  (*-- TRANSITION --------------------------------------------------------------------------------------------------------------*)
  (*-- working folder not existing ------------------------------------------------------*)
  IF (_Active = FALSE)
  THEN
    _DeleteState:= E_TraceDeleteStates.WaitFolder;
  (*-- delay time over ------------------------------------------------------------------*)
  ELSIF(F_GetTimeMsDiff(_DeleteTime) >= T#10S)
  THEN
    _DeleteState:= E_TraceDeleteStates.FolderStart;
  END_IF




(********************************************************************************************************************************)
(** prepare folder scan *********************************************************************************************************)
E_TraceDeleteStates.FolderStart:
  (*-- ENTRY -------------------------------------------------------------------------------------------------------------------*)
  IF (_DeleteStateLast <> _DeleteState)
  THEN
    _DeleteStateLast:= _DeleteState;
    _DeleteTime     := F_GetTimeMsTick();
    (*-- prepare folder scan ------------------------------------------------------------*)
    _ScanSubFolder.eCmd:= E_EnumCmdType.eEnumCmd_First;
  END_IF

  (*-- ACTION ------------------------------------------------------------------------------------------------------------------*)

  (*-- TRANSITION --------------------------------------------------------------------------------------------------------------*)
    _DeleteState:= E_TraceDeleteStates.FolderSeek;




(********************************************************************************************************************************)
(** find next (sub) folder ******************************************************************************************************)
E_TraceDeleteStates.FolderSeek:
  (*-- ENTRY -------------------------------------------------------------------------------------------------------------------*)
  IF (_DeleteStateLast <> _DeleteState)
  THEN
    _DeleteStateLast:= _DeleteState;
    _DeleteTime     := F_GetTimeMsTick();
    (*-----------------------------------------------------------------------------------*)
    _ScanSubFolder( bExecute:= FALSE );
    _ScanSubFolder.sNetID   := '';   // local
//  _ScanSubFolder.eCmd;   (* hier nicht beschreiben *)
    _ScanSubFolder.bExecute := TRUE;
    _ScanSubFolder.tTimeout := Tc2_System.DEFAULT_ADS_TIMEOUT;
    (*-----------------------------------------------------------------------------------*)
    DestStart:= ADR(_ScanSubFolder.sPathName);
    DestEnd  := ADR(_ScanSubFolder.sPathName) + SIZEOF(_ScanSubFolder.sPathName);
    DestStart:= F_StringCopy( DestStart:= DestStart,  DestEnd:= DestEnd,  Source:= ADR(_MainFolder)  );
    DestStart:= F_StringCopy( DestStart:= DestStart,  DestEnd:= DestEnd,  Source:= ADR('/*.*')  );
  END_IF

  (*-- ACTION ------------------------------------------------------------------------------------------------------------------*)
  _ScanSubFolder();

  (*-- TRANSITION --------------------------------------------------------------------------------------------------------------*)
  IF (_ScanSubFolder.bBusy = FALSE)
  THEN
    _ScanSubFolder.eCmd:= E_EnumCmdType.eEnumCmd_Next;
    (*-- error --------------------------------------------------------------------------*)
    IF    (_ScanSubFolder.bError = TRUE)
    THEN  (* unfortunately no difference between path noch found or destination not reachable *)
      _DeleteState:= E_TraceDeleteStates.WaitDelay;
    (*-- folder completely scanned ------------------------------------------------------*)
    ELSIF (_ScanSubFolder.bEOE = TRUE)
    THEN
      _DeleteState:= E_TraceDeleteStates.WaitDelay;
    (*-- found entry is no folder => continue -------------------------------------------*)
    ELSIF (_ScanSubFolder.stFindFile.fileAttributes.bDirectory = FALSE)
    THEN
      _DeleteStateLast:= E_TraceDeleteStates.Initialization;   // Re-entry
    (*-- folder name invalid => continue ------------------------------------------------*)
    ELSIF (    (_ScanSubFolder.stFindFile.sFileName = '.' )
            OR (_ScanSubFolder.stFindFile.sFileName = '..')  )
    THEN
      _DeleteStateLast:= E_TraceDeleteStates.Initialization;   // Re-entry
    (*-- folder valid => old enough to delete? ------------------------------------------*)
    ELSE
      (*-- parse folder name according to 'YYYY-MM-DD' --------------*)
      Result:= F_StringToTimeDate( AllowInvalidChars:= FALSE,  // invalid charachters will lead to parsing error
                                   DestStart        := ADR(_ScanSubFolder.stFindFile.sFileName),
                                   DestEnd          := ADR(_ScanSubFolder.stFindFile.sFileName) + SIZEOF(_ScanSubFolder.stFindFile.sFileName),
                                   Result     => FolderDate  );
      (*-- calc difference (in ms due to TIME limitation of 42d) ----*)
      SystemTimeTD:= SYSTEMTIME_TO_DT(System.fbSystemTime.TIMESTR);
      FolderTimeTD:= SYSTEMTIME_TO_DT(FolderDate);
      Diff_Seconds:= DT_TO_LINT(SystemTimeTD) - DT_TO_LINT(FolderTimeTD);
     (*-- folder name doesnt fit naming scheme YYYY-MM-DD -----------*)
      IF (Result = FALSE)
      THEN  // ignore ==> continue
        _DeleteStateLast:= E_TraceDeleteStates.Initialization;   // Re-entry
      (*-- folder from future ;-) -----------------------------------*)
      ELSIF (Diff_Seconds < 0)
      THEN  // ignore ==> continue
        _DeleteStateLast:= E_TraceDeleteStates.Initialization;   // Re-entry
      (*-- folder according parsed name too old ---------------------*)
      ELSIF (Diff_Seconds * 1_000 >= TIME_TO_LINT(SHELF_LIFE)  )  // TIME is internally already ms
      THEN  // => empty and delete
        _DeleteState:= E_TraceDeleteStates.FileStart;
      (*-- keep searching -------------------------------------------*)
      ELSE
        _DeleteStateLast:= E_TraceDeleteStates.Initialization;   // Re-entry
      END_IF
    END_IF
  END_IF




(********************************************************************************************************************************)
(** prepare file scan ***********************************************************************************************************)
E_TraceDeleteStates.FileStart:
  (*-- ENTRY -------------------------------------------------------------------------------------------------------------------*)
  IF (_DeleteStateLast <> _DeleteState)
  THEN
    _DeleteStateLast:= _DeleteState;
    _DeleteTime     := F_GetTimeMsTick();
    (*-----------------------------------------------------------------------------------*)
    _FileFind.eCmd:= E_EnumCmdType.eEnumCmd_First;
  END_IF

  (*-- ACTION ------------------------------------------------------------------------------------------------------------------*)

  (*-- TRANSITION --------------------------------------------------------------------------------------------------------------*)
  _DeleteState:= E_TraceDeleteStates.FileSeek;




(********************************************************************************************************************************)
(** find a file *****************************************************************************************************************)
E_TraceDeleteStates.FileSeek:
  (*-- ENTRY -------------------------------------------------------------------------------------------------------------------*)
  IF (_DeleteStateLast <> _DeleteState)
  THEN
    _DeleteStateLast:= _DeleteState;
    _DeleteTime     := F_GetTimeMsTick();
    (*-----------------------------------------------------------------------------------*)
    _FileFind( bExecute:= FALSE );
    _FileFind.sNetID   := '';   // local
//  _FileFind.eCmd;      (* hier nicht beschreiben *)
    _FileFind.bExecute := TRUE;
    _FileFind.tTimeout := Tc2_System.DEFAULT_ADS_TIMEOUT;
    (*-----------------------------------------------------------------------------------*)
    DestStart:= ADR(_FileFind.sPathName);
    DestEnd  := ADR(_FileFind.sPathName) + SIZEOF(_FileFind.sPathName);
    DestStart:= F_StringCopy( DestStart:= DestStart,  DestEnd:= DestEnd,  Source:= ADR(_MainFolder)  );
    DestStart:= F_StringCopy( DestStart:= DestStart,  DestEnd:= DestEnd,  Source:= ADR('/')  );
    DestStart:= F_StringCopy( DestStart:= DestStart,  DestEnd:= DestEnd,  Source:= ADR(_ScanSubFolder.stFindFile.sFileName)  );
    DestStart:= F_StringCopy( DestStart:= DestStart,  DestEnd:= DestEnd,  Source:= ADR('/*.*')  );
  END_IF

  (*-- ACTION ------------------------------------------------------------------------------------------------------------------*)
  _FileFind();

  (*-- TRANSITION --------------------------------------------------------------------------------------------------------------*)
  IF ( _FileFind.bBusy = FALSE )
  THEN
    _FileFind.eCmd:= E_EnumCmdType.eEnumCmd_Next;
    (*-- error --------------------------------------------------------------------------*)
    IF    (_FileFind.bError = TRUE)
    THEN
      _DeleteState:= E_TraceDeleteStates.WaitDelay;
    (*-- folder completely scanned ------------------------------------------------------*)
    ELSIF (_FileFind.bEOE = TRUE)
    THEN
      _DeleteState:= E_TraceDeleteStates.FolderDelete;
    (*-- file name invalid => continue --------------------------------------------------*)
    ELSIF (    (_FileFind.stFindFile.sFileName = '.' )
            OR (_FileFind.stFindFile.sFileName = '..')  )
    THEN
      _DeleteStateLast:= E_TraceDeleteStates.Initialization;   // Re-entry
    (*-- file found ==> delete ----------------------------------------------------------*)
    ELSE
      _DeleteState:= E_TraceDeleteStates.FileDelete;
    END_IF
  END_IF




(********************************************************************************************************************************)
(** delete this one file ********************************************************************************************************)
E_TraceDeleteStates.FileDelete:
  (*-- ENTRY -------------------------------------------------------------------------------------------------------------------*)
  IF (_DeleteStateLast <> _DeleteState)
  THEN
    _DeleteStateLast:= _DeleteState;
    _DeleteTime     := F_GetTimeMsTick();
    (*-----------------------------------------------------------------------------------*)
    _FileDelete( bExecute:= FALSE );
    _FileDelete.sNetId   := '';   // local
    _FileDelete.ePath    := E_OpenPath.PATH_GENERIC;  
    _FileDelete.bExecute := TRUE;
    _FileDelete.tTimeout := Tc2_System.DEFAULT_ADS_TIMEOUT;               
    (*-----------------------------------------------------------------------------------*)
    DestStart:= ADR(_FileDelete.sPathName);
    DestEnd  := ADR(_FileDelete.sPathName) + SIZEOF(_FileDelete.sPathName);
    DestStart:= F_StringCopy( DestStart:= DestStart,  DestEnd:= DestEnd,  Source:= ADR(_MainFolder)  );
    DestStart:= F_StringCopy( DestStart:= DestStart,  DestEnd:= DestEnd,  Source:= ADR('/')  );
    DestStart:= F_StringCopy( DestStart:= DestStart,  DestEnd:= DestEnd,  Source:= ADR(_ScanSubFolder.stFindFile.sFileName)  );
    DestStart:= F_StringCopy( DestStart:= DestStart,  DestEnd:= DestEnd,  Source:= ADR('/')  );
    DestStart:= F_StringCopy( DestStart:= DestStart,  DestEnd:= DestEnd,  Source:= ADR(_FileFind.stFindFile.sFileName)  );
  END_IF

  (*-- ACTION ------------------------------------------------------------------------------------------------------------------*)
  _FileDelete();

  (*-- TRANSITION --------------------------------------------------------------------------------------------------------------*)
  IF ( _FileDelete.bBusy = FALSE )
  THEN
    _DeleteState:= E_TraceDeleteStates.FileSeek;
  END_IF




(********************************************************************************************************************************)
(** delete that (now empty) folder **********************************************************************************************)
E_TraceDeleteStates.FolderDelete:
  (*-- ENTRY -------------------------------------------------------------------------------------------------------------------*)
  IF (_DeleteStateLast <> _DeleteState)
  THEN
    _DeleteStateLast:= _DeleteState;
    _DeleteTime     := F_GetTimeMsTick();
    (*-----------------------------------------------------------------------------------*)
    _FolderRemove( bExecute:= FALSE );
    _FolderRemove.sNetId   := '';   // local
    _FolderRemove.ePath    := E_OpenPath.PATH_GENERIC;
    _FolderRemove.bExecute := TRUE;
    _FolderRemove.tTimeout := Tc2_System.DEFAULT_ADS_TIMEOUT;
    (*-----------------------------------------------------------------------------------*)
    DestStart:= ADR(_FolderRemove.sPathName);
    DestEnd  := ADR(_FolderRemove.sPathName) + SIZEOF(_FolderRemove.sPathName);
    DestStart:= F_StringCopy( DestStart:= DestStart,  DestEnd:= DestEnd,  Source:= ADR(_MainFolder)  );
    DestStart:= F_StringCopy( DestStart:= DestStart,  DestEnd:= DestEnd,  Source:= ADR('/')  );
    DestStart:= F_StringCopy( DestStart:= DestStart,  DestEnd:= DestEnd,  Source:= ADR(_ScanSubFolder.stFindFile.sFileName)  );
    DestStart:= F_StringCopy( DestStart:= DestStart,  DestEnd:= DestEnd,  Source:= ADR('/')  );
  END_IF

  (*-- ACTION ------------------------------------------------------------------------------------------------------------------*)
  _FolderRemove();

  (*-- TRANSITION --------------------------------------------------------------------------------------------------------------*)
  IF ( _FolderRemove.bBusy = FALSE )
  THEN
    _DeleteState:= E_TraceDeleteStates.HddUsage;
    (*-- trace it ---------------------------------------------------*)
// example: '11-000-0000-00-0, old folder deleted,  folder = D:/Traces/1979-01-09/'
    _Text:= '';
    _Text:= CONCAT(_Text, F_AddDividerToSisString(SubsystemRegistry.SubsystemName) );
    _Text:= CONCAT(_Text, ',  old folder deleted');
    _Text:= CONCAT(_Text, DebugTextBlocks.FOLDER);
    _Text:= CONCAT(_Text, _FolderRemove.sPathName);
    Put( MsgType := E_DebugMsgType.INFO,
         Instance:= ADR(_Instance),
         Text    := ADR(_Text)  );
  END_IF




(********************************************************************************************************************************)
(** read current hdd usage ******************************************************************************************************)
E_TraceDeleteStates.HddUsage:
  (*-- ENTRY -------------------------------------------------------------------------------------------------------------------*)
  IF (_DeleteStateLast <> _DeleteState)
  THEN
    _DeleteStateLast:= _DeleteState;
    _DeleteTime     := F_GetTimeMsTick();
    (*-----------------------------------------------------------------------------------*)
    _HddUsage.Start( Drive:= _MainFolder );  // use drive letter from main folder
  END_IF

  (*-- ACTION ------------------------------------------------------------------------------------------------------------------*)

  (*-- TRANSITION --------------------------------------------------------------------------------------------------------------*)
  IF (_HddUsage.Busy = FALSE)
  THEN
    _HddUsageCount:= _HddUsageCount + 1;
    _HddStateLast := E_TraceHddUsageStates.Initialization;  // force re-entry and write message
    (*-------------------------------------------*)
    _DeleteState:= E_TraceDeleteStates.FolderSeek;
  END_IF




(********************************************************************************************************************************)
(** unknown *********************************************************************************************************************)
ELSE
  _DeleteState:= E_TraceDeleteStates.Initialization;
END_CASE




(********************************************************************************************************************************)
(** done ************************************************************************************************************************)
END_METHOD

// creates hdd usage debug messages
METHOD PROTECTED M_RunHddUsage

(********************************************************************************************************************************)
VAR
END_VAR

(********************************************************************************************************************************)
(** diagnosis *******************************************************************************************************************)
{warning disable C0139}
_HddUsage.BytesTotal;
_HddUsage.BytesUsed;    _HddUsage.PercentageUsed;
_HddUsage.BytesFree;    _HddUsage.PercentageFree;
{warning restore C0139}




(********************************************************************************************************************************)
(** initialisation **************************************************************************************************************)
CASE (_HddState) OF
E_TraceHddUsageStates.Initialization:
  (*-- ENTRY -------------------------------------------------------------------------------------------------------------------*)
    _HddStateLast:= _HddState;
    _HddTooFull  := FALSE;

  (*-- ACTION ------------------------------------------------------------------------------------------------------------------*)

  (*-- TRANSITION --------------------------------------------------------------------------------------------------------------*)
    // takes place in state E_TraceCheckStates.HddUsage of M_RunCheck()




(********************************************************************************************************************************)
(** unknown *********************************************************************************************************************)
E_TraceHddUsageStates.Unknown:
  (*-- ENTRY -------------------------------------------------------------------------------------------------------------------*)
  IF (_HddStateLast <> _HddState)
  THEN
    _HddStateLast:= _HddState;
    _HddTooFull  := FALSE;
    (*-----------------------------------------------------------------------------------*)
    // example: '11-000-0000-00-0, unable to retrieve hdd usage,  drive = D:/'
    _Text:= '';
    _Text:= CONCAT(_Text, F_AddDividerToSisString(SubsystemRegistry.SubsystemName) );
    _Text:= CONCAT(_Text, ',  unable to retrieve hdd usage');
    _Text:= CONCAT(_Text, DebugTextBlocks.DRIVE);
    _Text:= CONCAT(_Text, _HddUsage.Drive);
    IF (_HddFullMissed <> 0)
    THEN
      _Text:= CONCAT(_Text, DebugTextBlocks.MISSED);  _Text:= CONCAT(_Text, ULINT_TO_STRING(_HddFullMissed)   );
    END_IF
    Put( MsgType := E_DebugMsgType.ERROR,
         Instance:= ADR(_Instance),
         Text    := ADR(_Text)  );
    (*-----------------------------------------------------------------------------------*)
    _HddFullMissed:= 0;
  END_IF

  (*-- ACTION ------------------------------------------------------------------------------------------------------------------*)

  (*-- TRANSITION --------------------------------------------------------------------------------------------------------------*)
    // takes place in state E_TraceCheckStates.HddUsage of M_RunCheck()




(********************************************************************************************************************************)
(** enough space free ***********************************************************************************************************)
E_TraceHddUsageStates.EnoughFree:
  (*-- ENTRY -------------------------------------------------------------------------------------------------------------------*)
  IF (_HddStateLast <> _HddState)
  THEN
    _HddStateLast:= _HddState;
    _HddTooFull  := FALSE;
    (*-----------------------------------------------------------------------------------*)
    // example: '11-000-0000-00-0, hdd usage information,  drive = D:/:,  total = 320GB,  free = 98GB,  usage = 65%'
    _Text:= '';
    _Text:= CONCAT(_Text, F_AddDividerToSisString(SubsystemRegistry.SubsystemName) );
    _Text:= CONCAT(_Text, ',  hdd usage information');
    _Text:= CONCAT(_Text, DebugTextBlocks.DRIVE);  _Text:= CONCAT(_Text, _HddUsage.Drive);
    _Text:= CONCAT(_Text, DebugTextBlocks.TOTAL);  _Text:= CONCAT(_Text, F_DiskSpaceToString(_HddUsage.BytesTotal)  );
    _Text:= CONCAT(_Text, DebugTextBlocks.FREE);   _Text:= CONCAT(_Text, F_DiskSpaceToString(_HddUsage.BytesFree)   );
    _Text:= CONCAT(_Text, DebugTextBlocks.USED);   _Text:= CONCAT(_Text, F_DiskSpaceToString(_HddUsage.BytesUsed)   );
    _Text:= CONCAT(_Text, DebugTextBlocks.USAGE);  _Text:= CONCAT(_Text, BYTE_TO_STRING(_HddUsage.PercentageUsed)   );  _Text:= CONCAT(_Text, '%');
    IF (_HddFullMissed <> 0)
    THEN
      _Text:= CONCAT(_Text, DebugTextBlocks.MISSED);  _Text:= CONCAT(_Text, ULINT_TO_STRING(_HddFullMissed)   );
    END_IF
    Put( MsgType := E_DebugMsgType.INFO,
         Instance:= ADR(_Instance),
         Text    := ADR(_Text)  );
    (*-----------------------------------------------------------------------------------*)
    _HddFullMissed:= 0;
  END_IF

  (*-- ACTION ------------------------------------------------------------------------------------------------------------------*)

  (*-- TRANSITION --------------------------------------------------------------------------------------------------------------*)
    // takes place in state E_TraceCheckStates.HddUsage of M_RunCheck()




(********************************************************************************************************************************)
(** warning level ***************************************************************************************************************)
E_TraceHddUsageStates.WarningLevel:
  (*-- ENTRY -------------------------------------------------------------------------------------------------------------------*)
  IF (_HddStateLast <> _HddState)
  THEN
    _HddStateLast:= _HddState;
    _HddTooFull  := FALSE;
    (*-----------------------------------------------------------------------------------*)
    // example: '11-000-0000-00-0, hdd usage information,  drive = D:/:,  total = 320GB,  free = 98GB,  usage = 65%,  missed messages = 1234'
    _Text:= '';
    _Text:= CONCAT(_Text, F_AddDividerToSisString(SubsystemRegistry.SubsystemName) );
    _Text:= CONCAT(_Text, ',  hdd usage information');
    _Text:= CONCAT(_Text, DebugTextBlocks.DRIVE);  _Text:= CONCAT(_Text, _HddUsage.Drive);
    _Text:= CONCAT(_Text, DebugTextBlocks.TOTAL);  _Text:= CONCAT(_Text, F_DiskSpaceToString(_HddUsage.BytesTotal)  );
    _Text:= CONCAT(_Text, DebugTextBlocks.FREE);   _Text:= CONCAT(_Text, F_DiskSpaceToString(_HddUsage.BytesFree)   );
    _Text:= CONCAT(_Text, DebugTextBlocks.USED);   _Text:= CONCAT(_Text, F_DiskSpaceToString(_HddUsage.BytesUsed)   );
    _Text:= CONCAT(_Text, DebugTextBlocks.USAGE);  _Text:= CONCAT(_Text, BYTE_TO_STRING(_HddUsage.PercentageUsed)   );  _Text:= CONCAT(_Text, '%');
    IF (_HddFullMissed <> 0)
    THEN
      _Text:= CONCAT(_Text, DebugTextBlocks.MISSED);  _Text:= CONCAT(_Text, ULINT_TO_STRING(_HddFullMissed)   );
    END_IF
    Put( MsgType := E_DebugMsgType.WARNING,
         Instance:= ADR(_Instance),
         Text    := ADR(_Text)  );
    (*-----------------------------------------------------------------------------------*)
    _HddFullMissed:= 0;
  END_IF

  (*-- ACTION ------------------------------------------------------------------------------------------------------------------*)

  (*-- TRANSITION --------------------------------------------------------------------------------------------------------------*)
    // takes place in state E_TraceCheckStates.HddUsage of M_RunCheck()




(********************************************************************************************************************************)
(** error level *****************************************************************************************************************)
E_TraceHddUsageStates.ErrorLevel:
  (*-- ENTRY -------------------------------------------------------------------------------------------------------------------*)
  IF (_HddStateLast <> _HddState)
  THEN
    _HddStateLast:= _HddState;
    (*-----------------------------------------------------------------------------------*)
    // example: '11-000-0000-00-0, hdd usage information,  drive = D:/:,  total = 320GB,  free = 98GB,  usage = 65%'
    _Text:= '';
    _Text:= CONCAT(_Text, F_AddDividerToSisString(SubsystemRegistry.SubsystemName) );
    _Text:= CONCAT(_Text, ',  hdd usage information');
    _Text:= CONCAT(_Text, DebugTextBlocks.DRIVE);  _Text:= CONCAT(_Text, _HddUsage.Drive);
    _Text:= CONCAT(_Text, DebugTextBlocks.TOTAL);  _Text:= CONCAT(_Text, F_DiskSpaceToString(_HddUsage.BytesTotal)  );
    _Text:= CONCAT(_Text, DebugTextBlocks.FREE);   _Text:= CONCAT(_Text, F_DiskSpaceToString(_HddUsage.BytesFree)   );
    _Text:= CONCAT(_Text, DebugTextBlocks.USED);   _Text:= CONCAT(_Text, F_DiskSpaceToString(_HddUsage.BytesUsed)   );
    _Text:= CONCAT(_Text, DebugTextBlocks.USAGE);  _Text:= CONCAT(_Text, BYTE_TO_STRING(_HddUsage.PercentageUsed)   );  _Text:= CONCAT(_Text, '%');
    Put( MsgType := E_DebugMsgType.ERROR,
         Instance:= ADR(_Instance),
         Text    := ADR(_Text)  );
    (*-----------------------------------------------------------------------------------*)
    _HddTooFull   := TRUE; // after this Put() just above
    _HddFullMissed:= 0;
  END_IF

  (*-- ACTION ------------------------------------------------------------------------------------------------------------------*)

  (*-- TRANSITION --------------------------------------------------------------------------------------------------------------*)
    // takes place in state E_TraceCheckStates.HddUsage of M_RunCheck()




(********************************************************************************************************************************)
(** unknown *********************************************************************************************************************)
ELSE
  _HddState:= E_TraceHddUsageStates.Initialization;
END_CASE




(********************************************************************************************************************************)
(** done ************************************************************************************************************************)
END_METHOD

// writes traces into file
METHOD PROTECTED M_RunWrite

(********************************************************************************************************************************)
VAR
  DestStart             : POINTER TO BYTE                  := 0;     // start position to concat
  DestEnd               : POINTER TO BYTE                  := 0;     // buffer/string end
END_VAR

(********************************************************************************************************************************)
(** initialization **************************************************************************************************************)
CASE(_WriteState) OF
E_TraceWriteStates.Initialization:
  (*-- ENTRY -------------------------------------------------------------------------------------------------------------------*)
    _WriteStateLast:= _WriteState;

  (*-- ACTION ------------------------------------------------------------------------------------------------------------------*)

  (*-- TRANSITION --------------------------------------------------------------------------------------------------------------*)
  _WriteState:= E_TraceWriteStates.WaitFolder;




(********************************************************************************************************************************)
(** error - wait to disable *****************************************************************************************************)
E_TraceWriteStates.Error:
  (*-- ENTRY -------------------------------------------------------------------------------------------------------------------*)
  IF (_WriteStateLast <> _WriteState)
  THEN
    _WriteStateLast:= _WriteState;
    _WriteTime     := F_GetTimeMsTick();
    (*-----------------------------------------------------------------------------------*)
  END_IF

  (*-- ACTION ------------------------------------------------------------------------------------------------------------------*)

  (*-- TRANSITION --------------------------------------------------------------------------------------------------------------*)
  (*-- working folder dissapeared -------------------------------------------------------*)
  IF (_Active = FALSE)
  THEN
    _WriteState:= E_TraceWriteStates.WaitFolder;
  END_IF




(********************************************************************************************************************************)
(** wait working folder *********************************************************************************************************)
E_TraceWriteStates.WaitFolder:
  (*-- ENTRY -------------------------------------------------------------------------------------------------------------------*)
  IF (_WriteStateLast <> _WriteState)
  THEN
    _WriteStateLast:= _WriteState;
    _WriteTime     := F_GetTimeMsTick();
    (*-----------------------------------------------------------------------------------*)
  END_IF

  (*-- ACTION ------------------------------------------------------------------------------------------------------------------*)

  (*-- TRANSITION --------------------------------------------------------------------------------------------------------------*)
  (*-- working folder exists ------------------------------------------------------------*)
  IF (_Active = TRUE)
  THEN
    _WriteState:= E_TraceWriteStates.StartWork;
  END_IF




(********************************************************************************************************************************)
(** build working folder name with date *****************************************************************************************)
E_TraceWriteStates.StartWork:
  (*-- ENTRY -------------------------------------------------------------------------------------------------------------------*)
  IF (_WriteStateLast <> _WriteState)
  THEN
    _WriteStateLast:= _WriteState;
    _WriteTime     := F_GetTimeMsTick();
    (*-- save current working date ------------------------------------------------------*)
    _WriteDate:= System.fbSystemTime.TIMESTR;
    (*-- build folder name --------------------------------------------------------------*)
    DestStart:= ADR(_WritePath);
    DestEnd  := ADR(_WritePath) + SIZEOF(_WritePath);
    DestStart:= F_StringCopy          ( DestStart:= DestStart,  DestEnd:= DestEnd,  Source    := ADR(_MainFolder)  );
    DestStart:= F_StringCopy          ( DestStart:= DestStart,  DestEnd:= DestEnd,  Source    := ADR('/')  );
    DestStart:= F_StringFromDatestruct( DestStart:= DestStart,  DestEnd:= DestEnd,  DateStruct:= _WriteDate );
    DestStart:= F_StringCopy          ( DestStart:= DestStart,  DestEnd:= DestEnd,  Source    := ADR('/')  );
  END_IF

  (*-- ACTION ------------------------------------------------------------------------------------------------------------------*)

  (*-- TRANSITION --------------------------------------------------------------------------------------------------------------*)
  _WriteState:= E_TraceWriteStates.CreateDir;




(********************************************************************************************************************************)
(** create daily working folder *************************************************************************************************)
E_TraceWriteStates.CreateDir:
  (*-- ENTRY -------------------------------------------------------------------------------------------------------------------*)
  IF (_WriteStateLast <> _WriteState)
  THEN
    _WriteStateLast:= _WriteState;
    _WriteTime     := F_GetTimeMsTick();
    (*-----------------------------------------------------------------------------------*)
    _CreateDir( bExecute:= FALSE );         
    _CreateDir.sNetId   := '';  // local
    _CreateDir.sPathName:= _WritePath;
    _CreateDir.ePath    := E_OpenPath.PATH_GENERIC;
    _CreateDir.bExecute := TRUE;         
    _CreateDir.tTimeout := Tc2_System.DEFAULT_ADS_TIMEOUT;
  END_IF

  (*-- ACTION ------------------------------------------------------------------------------------------------------------------*)
  _CreateDir();

  (*-- TRANSITION --------------------------------------------------------------------------------------------------------------*)
  IF (_CreateDir.bBusy = FALSE)
  THEN
    (*-- folder created => continue -----------------------------------------------------*)
    IF ( _CreateDir.bError = FALSE )
    THEN
      _WriteState:= E_TraceWriteStates.ScanFileStart;
      (*-- trace it -------------------------------------------------*)
// example: '11-000-0000-00-0, new folder created,  folder = D:/Traces/1979-01-09/'
      _Text:= '';
      _Text:= CONCAT(_Text, F_AddDividerToSisString(SubsystemRegistry.SubsystemName) );
      _Text:= CONCAT(_Text, ',  new folder created');
      _Text:= CONCAT(_Text, DebugTextBlocks.FOLDER);
      _Text:= CONCAT(_Text, _CreateDir.sPathName);
      Put( MsgType := E_DebugMsgType.INFO,
           Instance:= ADR(_Instance),
           Text    := ADR(_Text)  );
    (*-- folder already exists ----------------------------------------------------------*)
    ELSIF (    ( _CreateDir.nErrId = 16#070C )     // ADSERR_DEVICE_NOTFOUND
            OR ( _CreateDir.nErrId = 16#0723 )  )  // ADSERR_DEVICE_ACCESSDENIED
    THEN                                           // BKF-Flick: Änderung der ReturnCodes ab 4022.20
      _WriteState:= E_TraceWriteStates.ScanFileStart;
    (*-- error --------------------------------------------------------------------------*)
    ELSE
      _WriteState:= E_TraceWriteStates.Error;
    END_IF
  END_IF




(********************************************************************************************************************************)
(** prepare folder scan for existing files **************************************************************************************)
E_TraceWriteStates.ScanFileStart:
  (*-- ENTRY -------------------------------------------------------------------------------------------------------------------*)
  IF (_WriteStateLast <> _WriteState)
  THEN
    _WriteStateLast:= _WriteState;
    _WriteTime     := F_GetTimeMsTick();
    (*-----------------------------------------------------------------------------------*)
    _FileIndex     := 1;  (* Filenummerierung beginnt bei Eins *)
    _FileCheck.eCmd:= eEnumCmd_First;
  END_IF

  (*-- ACTION ------------------------------------------------------------------------------------------------------------------*)

  (*-- TRANSITION --------------------------------------------------------------------------------------------------------------*)
    _WriteState:= E_TraceWriteStates.ScanFileExists;




(********************************************************************************************************************************)
(** scan folder to check if files exist? ****************************************************************************************)
E_TraceWriteStates.ScanFileExists:
  (*-- ENTRY -------------------------------------------------------------------------------------------------------------------*)
  IF (_WriteStateLast <> _WriteState)
  THEN
    _WriteStateLast:= _WriteState;
    _WriteTime     := F_GetTimeMsTick();
    (*-- build file name with _FileIndex ------------------------------------------------*)
{warning disable C0139}
    M_BuildFileName();    _WriteFileName;
{warning restore C0139}
   (*-----------------------------------------------------------------------------------*)
    _FileCheck( bExecute:= FALSE );
    _FileCheck.sNetID   := '';  // local
//  _FileCheck.eCmd;   // maintain this value here 
    _FileCheck.bExecute := TRUE;
    _FileCheck.tTimeout := Tc2_System.DEFAULT_ADS_TIMEOUT;
    (*-----------------------------------------------------------------------------------*)
    DestStart:= ADR(_FileCheck.sPathName);
    DestEnd  := ADR(_FileCheck.sPathName) + SIZEOF(_FileCheck.sPathName);
    DestStart:= F_StringCopy( DestStart:= DestStart,  DestEnd:= DestEnd,  Source:= ADR(_WritePath)  );
    DestStart:= F_StringCopy( DestStart:= DestStart,  DestEnd:= DestEnd,  Source:= ADR(_WriteFileName)  );
  END_IF

  (*-- ACTION ------------------------------------------------------------------------------------------------------------------*)
  _FileCheck();

  (*-- TRANSITION --------------------------------------------------------------------------------------------------------------*)
  IF (_FileCheck.bBusy = FALSE)
  THEN
    _FileCheck.eCmd:= E_EnumCmdType.eEnumCmd_Next;
    (*-- error --------------------------------------------------------------------------*)
    IF ( _FileCheck.bError = TRUE )
    THEN
      _WriteState:= E_TraceWriteStates.Error;
    (*-- index does not exist => create & use -------------------------------------------*)
    ELSIF ( _FileCheck.bEOE = TRUE )
    THEN
      _WriteState:= E_TraceWriteStates.CreateOpen;
    (*-- found: but already too large => keep searching ---------------------------------*)
    ELSIF (    (_FileCheck.stFindFile.fileSize.dwLowPart)
            >= (_MaxFileSizeKB * DWORD#1024             )   ) (* kilo bytes => bytes *)
    THEN
      _WriteState:= E_TraceWriteStates.ScanFileCancel;
    (*-- found: smaller than max size => keep using -------------------------------------*)
    ELSE
      _WriteState:= E_TraceWriteStates.ScanFileAbort;
    END_IF
  END_IF




(********************************************************************************************************************************)
(** cancel scan *****************************************************************************************************************)
E_TraceWriteStates.ScanFileCancel:
  (*-- ENTRY -------------------------------------------------------------------------------------------------------------------*)
  IF (_WriteStateLast <> _WriteState)
  THEN
    _WriteStateLast:= _WriteState;
    _WriteTime     := F_GetTimeMsTick();
    (*-----------------------------------------------------------------------------------*)
    _FileCheck( bExecute:= FALSE );
    _FileCheck.sNetID   := '';  // local
//  _FileCheck.sPathName;  // maintain this value here 
    _FileCheck.eCmd     := E_EnumCmdType.eEnumCmd_Abort;
    _FileCheck.bExecute := TRUE;
    _FileCheck.tTimeout := Tc2_System.DEFAULT_ADS_TIMEOUT;
  END_IF

  (*-- ACTION ------------------------------------------------------------------------------------------------------------------*)
  _FileCheck();

  (*-- TRANSITION --------------------------------------------------------------------------------------------------------------*)
  IF (_FileCheck.bBusy = FALSE)
  THEN
    (*-- error --------------------------------------------------------------------------*)
    IF ( _FileCheck.bError = TRUE )
    THEN
      _WriteState:= E_TraceWriteStates.Error;
    (*-- cancellation successful --------------------------------------------------------*)
    ELSIF ( _FileCheck.bEOE = TRUE )
    THEN
      _FileIndex     := _FileIndex + 1;
      _FileCheck.eCmd:= eEnumCmd_First;
      _WriteState    := E_TraceWriteStates.ScanFileExists;
    (*-- keep searching -----------------------------------------------------------------*)
    ELSE
      _WriteStateLast:= E_TraceWriteStates.Initialization;  // Re-entry
    END_IF
  END_IF




(********************************************************************************************************************************)
(** cancel scan *****************************************************************************************************************)
E_TraceWriteStates.ScanFileAbort:
  (*-- ENTRY -------------------------------------------------------------------------------------------------------------------*)
  IF (_WriteStateLast <> _WriteState)
  THEN
    _WriteStateLast:= _WriteState;
    _WriteTime     := F_GetTimeMsTick();
    (*-----------------------------------------------------------------------------------*)
    _FileCheck( bExecute:= FALSE );
    _FileCheck.sNetID   := '';  // local
//  _FileCheck.sPathName;  // maintain this value here 
    _FileCheck.eCmd     := E_EnumCmdType.eEnumCmd_Abort;
    _FileCheck.bExecute := TRUE;
    _FileCheck.tTimeout := Tc2_System.DEFAULT_ADS_TIMEOUT;
  END_IF

  (*-- ACTION ------------------------------------------------------------------------------------------------------------------*)
  _FileCheck();

  (*-- TRANSITION --------------------------------------------------------------------------------------------------------------*)
  IF (_FileCheck.bBusy = FALSE)
  THEN
    (*-- error --------------------------------------------------------------------------*)
    IF    ( _FileCheck.bError = TRUE )
    THEN
      _WriteState:= E_TraceWriteStates.Error;
    (*-- cancellation successful --------------------------------------------------------*)
    ELSIF ( _FileCheck.bEOE = TRUE )
    THEN
      _WriteState:= E_TraceWriteStates.WaitForTrace;
    (*-- keep searching -----------------------------------------------------------------*)
    ELSE                                     
      _WriteStateLast:= E_TraceWriteStates.Initialization;  // Re-entry
    END_IF
  END_IF




(********************************************************************************************************************************)
(** create new file *************************************************************************************************************)
E_TraceWriteStates.CreateOpen:
  (*-- ENTRY -------------------------------------------------------------------------------------------------------------------*)
  IF (_WriteStateLast <> _WriteState)
  THEN
    _WriteStateLast:= _WriteState;
    _WriteTime     := F_GetTimeMsTick();
    (*-- build file name with _FileIndex ------------------------------------------------*)
{warning disable C0139}
    M_BuildFileName();    _WriteFileName;
{warning restore C0139}
    (*-----------------------------------------------------------------------------------*)
    _FileOpen( bExecute:= FALSE );
    _FileOpen.sNetId   := '';  // local
    _FileOpen.nMode    := ( FOPEN_MODEWRITE OR FOPEN_MODEPLUS OR FOPEN_MODEBINARY );
    _FileOpen.ePath    := E_OpenPath.PATH_GENERIC;          
    _FileOpen.bExecute := TRUE;
    _FileOpen.tTimeout := Tc2_System.DEFAULT_ADS_TIMEOUT;
    (*-----------------------------------------------------------------------------------*)
    DestStart:= ADR(_FileOpen.sPathName);
    DestEnd  := ADR(_FileOpen.sPathName) + SIZEOF(_FileOpen.sPathName);
    DestStart:= F_StringCopy( DestStart:= DestStart,  DestEnd:= DestEnd,  Source:= ADR(_WritePath)  );
    DestStart:= F_StringCopy( DestStart:= DestStart,  DestEnd:= DestEnd,  Source:= ADR(_WriteFileName)  );
  END_IF

  (*-- ACTION ------------------------------------------------------------------------------------------------------------------*)
  _FileOpen();

  (*-- TRANSITION --------------------------------------------------------------------------------------------------------------*)
  IF (_FileOpen.bBusy = FALSE)
  THEN
    (*-- File angelegt ------------------------------------------------------------------*)
    IF    ( _FileOpen.bError = FALSE )  
    THEN
      _Statistics.FileOpenCounter:= _Statistics.FileOpenCounter + 1;
      (*-----------------------------------------*)
      _Opened        := TRUE;
      _FileTimeOpened:= F_GetTimeMsTick();
      _WriteState    := E_TraceWriteStates.CreateHeader;
   (*-- folder doesn't exist (anymore) --------------------------------------------------*)
    ELSIF ( _FileOpen.nErrId = 16#070C )
    THEN
      _WriteState:= E_TraceWriteStates.StartWork;    
    (*-- error --------------------------------------------------------------------------*)
    ELSE
      _WriteState:= E_TraceWriteStates.Error;
    END_IF
  END_IF




(********************************************************************************************************************************)
(** write header ****************************************************************************************************************)
E_TraceWriteStates.CreateHeader:
  (*-- ENTRY -------------------------------------------------------------------------------------------------------------------*)
  IF (_WriteStateLast <> _WriteState)
  THEN
    _WriteStateLast:= _WriteState;
    _WriteTime     := F_GetTimeMsTick();
    (*-- create file header -------------------------------------------------------------*)
{warning disable C0139}
    M_CreateHeader();   _DataLength;
{warning restore C0139}
    (*-----------------------------------------------------------------------------------*)
    _FileWrite( bExecute:= FALSE );
    _FileWrite.sNetId    := '';  // local               
    _FileWrite.hFile     := _FileOpen.hFile;       
    _FileWrite.pWriteBuff:= ADR(_DataBuffer);
    _FileWrite.cbWriteLen:= _DataLength;
    _FileWrite.bExecute  := TRUE;
    _FileWrite.tTimeout  := Tc2_System.DEFAULT_ADS_TIMEOUT;
  END_IF

  (*-- ACTION ------------------------------------------------------------------------------------------------------------------*)
  _FileWrite();

  (*-- TRANSITION --------------------------------------------------------------------------------------------------------------*)
  IF (_FileWrite.bBusy = FALSE)
  THEN
    (*-- error --------------------------------------------------------------------------*)
    IF    ( _FileWrite.bError = TRUE )
    THEN
      _WriteState:= E_TraceWriteStates.Error;
    (*-- writing successful -------------------------------------------------------------*)
    ELSE
      _WriteState:= E_TraceWriteStates.CreateClose;
    END_IF
  END_IF




(********************************************************************************************************************************)
(** close new file **************************************************************************************************************)
E_TraceWriteStates.CreateClose:
  (*-- ENTRY -------------------------------------------------------------------------------------------------------------------*)
  IF (_WriteStateLast <> _WriteState)
  THEN
    _WriteStateLast:= _WriteState;
    _WriteTime     := F_GetTimeMsTick();
    (*-----------------------------------------------------------------------------------*)
    _FileClose( bExecute:= FALSE );
    _FileClose.sNetId  := '';   // local
    _FileClose.hFile   := _FileOpen.hFile;
    _FileClose.bExecute:= TRUE;
    _FileClose.tTimeout:= Tc2_System.DEFAULT_ADS_TIMEOUT;
  END_IF

  (*-- ACTION ------------------------------------------------------------------------------------------------------------------*)
  _FileClose();

  (*-- TRANSITION --------------------------------------------------------------------------------------------------------------*)
  IF (_FileClose.bBusy = FALSE)
  THEN
    _PlcRestarted:= FALSE;
    _Opened      := FALSE;
    (*-- calculate maximum file open time -----------------------------------------------*)
    _Statistics.MaxFileOpenTime:= MAX( _Statistics.MaxFileOpenTime, F_GetTimeMsDiff(_FileTimeOpened)  );
    (*-- error --------------------------------------------------------------------------*)
    IF    ( _FileClose.bError = TRUE )
    THEN
      _WriteState:= E_TraceWriteStates.Error;
    (*-- closing successful -------------------------------------------------------------*)
    ELSE
      _WriteState:= E_TraceWriteStates.WaitForTrace;
    END_IF
  END_IF




(********************************************************************************************************************************)
(** inhibit time (currently not used) *******************************************************************************************)
E_TraceWriteStates.WaitLocked:
  (*-- ENTRY -------------------------------------------------------------------------------------------------------------------*)
  IF (_WriteStateLast <> _WriteState)
  THEN
    _WriteStateLast:= _WriteState;
    _WriteTime     := F_GetTimeMsTick();
    (*-----------------------------------------------------------------------------------*)
  END_IF

  (*-- ACTION ------------------------------------------------------------------------------------------------------------------*)

  (*-- TRANSITION --------------------------------------------------------------------------------------------------------------*)
  (*-- (still) too many traces to be written -> skip inhibit time -----------------------*)
  IF (_FifoFillLevel >= 256)
  THEN
    _WriteState:= E_TraceWriteStates.WaitForTrace;
  (*-- inhibit time over ----------------------------------------------------------------*)
  ELSIF (F_GetTimeMsDiff(_WriteTime) >= LOCKTIME)
  THEN
    _WriteState:= E_TraceWriteStates.WaitForTrace;
  (*-- working folder dissapeared -------------------------------------------------------*)
  ELSIF (_Active = FALSE)
  THEN
    _WriteState:= E_TraceWriteStates.WaitFolder;
  END_IF




(********************************************************************************************************************************)
(** idle -> wait for traces to write ********************************************************************************************)
E_TraceWriteStates.WaitForTrace:
  (*-- ENTRY -------------------------------------------------------------------------------------------------------------------*)
  IF (_WriteStateLast <> _WriteState)
  THEN
    _WriteStateLast:= _WriteState;
    _WriteTime     := F_GetTimeMsTick();
    (*-----------------------------------------------------------------------------------*)
  END_IF

  (*-- ACTION ------------------------------------------------------------------------------------------------------------------*)

  (*-- TRANSITION --------------------------------------------------------------------------------------------------------------*)
  (*-- traces to write available --------------------------------------------------------*)
  IF (_FifoFillLevel <> 0)
  THEN
//  IF ( _FileIndex <> 1 ) 
//  THEN
//     => check if file-one (still) exists
//  ELSE
    _FileCheck.eCmd:= E_EnumCmdType.eEnumCmd_First;
    _WriteState    := E_TraceWriteStates.FileSizeExists;
  (*-- working folder dissapeared -------------------------------------------------------*)
  ELSIF (_Active = FALSE)
  THEN
    _WriteState:= E_TraceWriteStates.WaitFolder;
  END_IF




(********************************************************************************************************************************)
(** check if current file (_FileIndex) still exists and if it's (already) too large *********************************************)
E_TraceWriteStates.FileSizeExists:
  (*-- ENTRY -------------------------------------------------------------------------------------------------------------------*)
  IF (_WriteStateLast <> _WriteState)
  THEN
    _WriteStateLast:= _WriteState;
    _WriteTime     := F_GetTimeMsTick();
    (*-----------------------------------------------------------------------------------*)
    _FileCheck( bExecute:= FALSE );
    _FileCheck.sNetID   := '';   // local
//  _FileCheck.eCmd;   (* nicht beschreiben *)
    _FileCheck.bExecute := TRUE;
    _FileCheck.tTimeout := Tc2_System.DEFAULT_ADS_TIMEOUT;
    (*-----------------------------------------------------------------------------------*)
    DestStart:= ADR(_FileCheck.sPathName);
    DestEnd  := ADR(_FileCheck.sPathName) + SIZEOF(_FileCheck.sPathName);
    DestStart:= F_StringCopy( DestStart:= DestStart,  DestEnd:= DestEnd,  Source:= ADR(_WritePath)  );
    DestStart:= F_StringCopy( DestStart:= DestStart,  DestEnd:= DestEnd,  Source:= ADR(_WriteFileName)  );
  END_IF

  (*-- ACTION ------------------------------------------------------------------------------------------------------------------*)
  _FileCheck();

  (*-- TRANSITION --------------------------------------------------------------------------------------------------------------*)
  IF (_FileCheck.bBusy = FALSE)
  THEN
    (*-- error --------------------------------------------------------------------------*)
    IF    (_FileCheck.bError = TRUE)
    THEN
      _WriteState:= E_TraceWriteStates.Error;
    (*-- doesnt exists (anymore) => rescan ----------------------------------------------*)
    ELSIF (_FileCheck.bEOE = TRUE)
    THEN
      _WriteState:= E_TraceWriteStates.ScanFileStart;
    (*-- exists: => use it --------------------------------------------------------------*)
    ELSE
      _FileSize  := (        DWORD_TO_ULINT(_FileCheck.stFindFile.fileSize.dwLowPart )
                      OR SHL(DWORD_TO_ULINT(_FileCheck.stFindFile.fileSize.dwHighPart), 32)  );
      (*-- maximal file size exceeded -----------*)
      IF (    (_FileSize (* KiloBytes => Bytes *) )
           >= (_MaxFileSizeKB * ULINT#1024        )   )  THEN   _WriteState:= E_TraceWriteStates.FileSizeCancel;  // start over with new file index
      ELSE                                                      _WriteState:= E_TraceWriteStates.FileSizeAbort;   // use this file again
      END_IF
    END_IF
  END_IF




(********************************************************************************************************************************)
(** cancel file size/exist check and use this ***********************************************************************************)
E_TraceWriteStates.FileSizeAbort:
  (*-- ENTRY -------------------------------------------------------------------------------------------------------------------*)
  IF (_WriteStateLast <> _WriteState)
  THEN
    _WriteStateLast:= _WriteState;
    _WriteTime     := F_GetTimeMsTick();
    (*-----------------------------------------------------------------------------------*)
    _FileCheck( bExecute:= FALSE );
    _FileCheck.sNetID   := '';   // local
//  _FileCheck.sPathName;  remain value
    _FileCheck.eCmd     := E_EnumCmdType.eEnumCmd_Abort;
    _FileCheck.bExecute := TRUE;
    _FileCheck.tTimeout := Tc2_System.DEFAULT_ADS_TIMEOUT;
  END_IF

  (*-- ACTION ------------------------------------------------------------------------------------------------------------------*)
  _FileCheck();

  (*-- TRANSITION --------------------------------------------------------------------------------------------------------------*)
  IF ( _FileCheck.bBusy = FALSE )
  THEN
    (*-- error --------------------------------------------------------------------------*)
    IF    (_FileCheck.bError = TRUE)
    THEN
      _WriteState:= E_TraceWriteStates.Error;
    (*-- finished -----------------------------------------------------------------------*)
    ELSIF (_FileCheck.bEOE = TRUE)
    THEN
      _WriteState:= E_TraceWriteStates.OpenAppend;
    (*-- keep searching -----------------------------------------------------------------*)
    ELSE
      _WriteStateLast:= E_TraceWriteStates.Initialization;  // Re-entry
    END_IF
  END_IF



(********************************************************************************************************************************)
(** cancel file size/exist check due to file size already too large *************************************************************)
E_TraceWriteStates.FileSizeCancel:
  (*-- ENTRY -------------------------------------------------------------------------------------------------------------------*)
  IF (_WriteStateLast <> _WriteState)
  THEN
    _WriteStateLast:= _WriteState;
    _WriteTime     := F_GetTimeMsTick();
    (*-----------------------------------------------------------------------------------*)
    _FileCheck( bExecute:= FALSE );
    _FileCheck.sNetID   := '';   // local
//  _FileCheck.sPathName;  remain value
    _FileCheck.eCmd     := E_EnumCmdType.eEnumCmd_Abort;
    _FileCheck.bExecute := TRUE;
    _FileCheck.tTimeout := Tc2_System.DEFAULT_ADS_TIMEOUT;
  END_IF

  (*-- ACTION ------------------------------------------------------------------------------------------------------------------*)
  _FileCheck();

  (*-- TRANSITION --------------------------------------------------------------------------------------------------------------*)
  IF ( _FileCheck.bBusy = FALSE )
  THEN
    (*-- error --------------------------------------------------------------------------*)
    IF    (_FileCheck.bError = TRUE)
    THEN
      _WriteState:= E_TraceWriteStates.Error;
    (*-- finished -----------------------------------------------------------------------*)
    ELSIF (_FileCheck.bEOE = TRUE)
    THEN
      _FileIndex := _FileIndex + 1;
      _WriteState:= E_TraceWriteStates.CreateOpen;
    (*-- keep searching -----------------------------------------------------------------*)
    ELSE
      _WriteStateLast:= E_TraceWriteStates.Initialization;  // Re-entry
    END_IF
  END_IF




(********************************************************************************************************************************)
(** open file to write/append ***************************************************************************************************)
E_TraceWriteStates.OpenAppend:
  (*-- ENTRY -------------------------------------------------------------------------------------------------------------------*)
  IF (_WriteStateLast <> _WriteState)
  THEN
    _WriteStateLast:= _WriteState;
    _WriteTime     := F_GetTimeMsTick();
    (*-----------------------------------------------------------------------------------*)
    _FileOpen( bExecute:= FALSE );
    _FileOpen.sNetId   := '';   // local
    _FileOpen.nMode    := ( FOPEN_MODEAPPEND OR FOPEN_MODEBINARY );                                
    _FileOpen.ePath    := E_OpenPath.PATH_GENERIC;          
    _FileOpen.bExecute := TRUE;
    _FileOpen.tTimeout := Tc2_System.DEFAULT_ADS_TIMEOUT;
    (*-----------------------------------------------------------------------------------*)
    DestStart:= ADR(_FileOpen.sPathName);
    DestEnd  := ADR(_FileOpen.sPathName) + SIZEOF(_FileOpen.sPathName);
    DestStart:= F_StringCopy( DestStart:= DestStart,  DestEnd:= DestEnd,  Source:= ADR(_WritePath)  );
    DestStart:= F_StringCopy( DestStart:= DestStart,  DestEnd:= DestEnd,  Source:= ADR(_WriteFileName)  );
  END_IF

  (*-- ACTION ------------------------------------------------------------------------------------------------------------------*)
  _FileOpen();

  (*-- TRANSITION --------------------------------------------------------------------------------------------------------------*)
  IF ( _FileOpen.bBusy = FALSE )
  THEN
    (*-- file opened --------------------------------------------------------------------*)
    IF    ( _FileOpen.bError = FALSE )  
    THEN
      _Statistics.FileOpenCounter:= _Statistics.FileOpenCounter + 1;
      _FileTimeOpened            := F_GetTimeMsTick();
      _Opened                    := TRUE;
      (*-----------------------------------------*)
      IF (_PlcRestarted = TRUE) THEN   _WriteState:= E_TraceWriteStates.WriteDivider;
      ELSE                             _WriteState:= E_TraceWriteStates.WriteData;
      END_IF
    (*-- folder doesn't exist (anymore) -------------------------------------------------*)
    ELSIF ( _FileOpen.nErrId = 16#070C )
    THEN
      _WriteState:= E_TraceWriteStates.StartWork;    
    (*-- error --------------------------------------------------------------------------*)
    ELSE
      _WriteState:= E_TraceWriteStates.Error;
    END_IF
  END_IF




(********************************************************************************************************************************)
(** add plc restart divider *****************************************************************************************************)
E_TraceWriteStates.WriteDivider:
  (*-- ENTRY -------------------------------------------------------------------------------------------------------------------*)
  IF (_WriteStateLast <> _WriteState)
  THEN
    _WriteStateLast:= _WriteState;
    _WriteTime     := F_GetTimeMsTick();
    (*-- create plc divider -------------------------------------------------------------*)
{warning disable C0139}
    M_CreatePlcDivider();   _DataLength;
{warning restore C0139}
    (*-----------------------------------------------------------------------------------*)
    _FileWrite( bExecute:= FALSE );
    _FileWrite.sNetId    := '';  // local               
    _FileWrite.hFile     := _FileOpen.hFile;       
    _FileWrite.pWriteBuff:= ADR(_DataBuffer);
    _FileWrite.cbWriteLen:= _DataLength;
    _FileWrite.bExecute  := TRUE;
    _FileWrite.tTimeout  := Tc2_System.DEFAULT_ADS_TIMEOUT;
  END_IF

  (*-- ACTION ------------------------------------------------------------------------------------------------------------------*)
  _FileWrite();

  (*-- TRANSITION --------------------------------------------------------------------------------------------------------------*)
  IF (_FileWrite.bBusy = FALSE)
  THEN
    _PlcRestarted:= FALSE;
    _FileSize    := _FileSize + _FileWrite.cbWrite;
    (*-- error --------------------------------------------------------------------------*)
    IF    (_FileWrite.bError = TRUE)
    THEN
      _WriteState:= E_TraceWriteStates.CloseOpenTime;
    (*-- writing successful -------------------------------------------------------------*)
    ELSE
      _WriteState:= E_TraceWriteStates.WriteData;
    END_IF
  END_IF




(********************************************************************************************************************************)
(** write trace lines ***********************************************************************************************************)
E_TraceWriteStates.WriteData:
  (*-- ENTRY -------------------------------------------------------------------------------------------------------------------*)
  IF (_WriteStateLast <> _WriteState)
  THEN
    _WriteStateLast:= _WriteState;
    _WriteTime     := F_GetTimeMsTick();
    (*-- create data --------------------------------------------------------------------*)
{warning disable C0139}
    _DataDateChanged:= M_CreateData();   _DataLength;
    (*-----------------------------------------------------------------------------------*)
    _FileWrite( bExecute:= FALSE );
    _FileWrite.sNetId    := '';  // local               
    _FileWrite.hFile     := _FileOpen.hFile;       
    _FileWrite.pWriteBuff:= ADR(_DataBuffer);
    _FileWrite.cbWriteLen:= _DataLength;
    _FileWrite.bExecute  := TRUE;
    _FileWrite.tTimeout  := Tc2_System.DEFAULT_ADS_TIMEOUT;
{warning restore C0139}
  END_IF

  (*-- ACTION ------------------------------------------------------------------------------------------------------------------*)
  _FileWrite();

  (*-- TRANSITION --------------------------------------------------------------------------------------------------------------*)
  IF ( _FileWrite.bBusy = FALSE )
  THEN
    _FileSize:= _FileSize + _FileWrite.cbWrite;
    (*-- error --------------------------------------------------------------------------*)
    IF    (_FileWrite.bError = TRUE)
    THEN
      _WriteState:= E_TraceWriteStates.CloseOpenTime;
    (*-- trace date changed -> new date folder ------------------------------------------*)
    ELSIF (_DataDateChanged = TRUE)
    THEN  (* new file/folder for new day *)
      _WriteState:= E_TraceWriteStates.EofDate;
    (*-- maximum file size exceeded -----------------------------------------------------*)
    ELSIF (    (_FileSize (* KiloBytes => Bytes *) )
            >= (_MaxFileSizeKB * ULINT#1024        )   )
    THEN  (* start over with new file index *)
      _WriteState:= E_TraceWriteStates.EofSize;
    (*-- maximum file open time exceeded (flush) ----------------------------------------*)
    ELSIF (F_GetTimeMsDiff(_FileTimeOpened) >= MAX_FILEOPEN_TIME)
    THEN  (* close file and re-open it => file flush *)
      _WriteState:= E_TraceWriteStates.CloseOpenTime;
    (*-- more to write? -----------------------------------------------------------------*)
    ELSIF (_FifoFillLevel <> 0)
    THEN
      _WriteStateLast:= E_TraceWriteStates.Initialization;  // Re-entry
    (*-- no traces to write anymore -> close & wait -------------------------------------*)
    ELSE
      _WriteState:= E_TraceWriteStates.CloseOpenTime;
    END_IF
  END_IF




(********************************************************************************************************************************)
(** close due to max open time exceeded *****************************************************************************************)
E_TraceWriteStates.CloseOpenTime:
  (*-- ENTRY -------------------------------------------------------------------------------------------------------------------*)
  IF (_WriteStateLast <> _WriteState)
  THEN
    _WriteStateLast:= _WriteState;
    _WriteTime     := F_GetTimeMsTick();
    (*-----------------------------------------------------------------------------------*)
    _FileClose( bExecute:= FALSE );
    _FileClose.sNetId  := '';  // local
    _FileClose.hFile   := _FileOpen.hFile;
    _FileClose.bExecute:= TRUE;
    _FileClose.tTimeout:= Tc2_System.DEFAULT_ADS_TIMEOUT;
  END_IF

  (*-- ACTION ------------------------------------------------------------------------------------------------------------------*)
  _FileClose();

  (*-- TRANSITION --------------------------------------------------------------------------------------------------------------*)
  IF (_FileClose.bBusy = FALSE)
  THEN
    _Opened:= FALSE;
    (*-- calculate maximum file open time -----------------------------------------------*)
    _Statistics.MaxFileOpenTime:= MAX( _Statistics.MaxFileOpenTime, F_GetTimeMsDiff(_FileTimeOpened)  );
    (*-- error --------------------------------------------------------------------------*)
    IF    (_FileClose.bError = TRUE)
    THEN
      _WriteState:= E_TraceWriteStates.Error;
    (*-- closing successful -------------------------------------------------------------*)
    ELSE
      _WriteState:= E_TraceWriteStates.WaitLocked;
    END_IF
  END_IF




(********************************************************************************************************************************)
(** add eof due max file size exceeded ******************************************************************************************)
E_TraceWriteStates.EofSize:
  (*-- ENTRY -------------------------------------------------------------------------------------------------------------------*)
  IF (_WriteStateLast <> _WriteState)
  THEN
    _WriteStateLast:= _WriteState;
    _WriteTime     := F_GetTimeMsTick();
    (*-- create eof ---------------------------------------------------------------------*)
{warning disable C0139}
    M_CreateEof();   _DataLength;
{warning restore C0139}
    (*-----------------------------------------------------------------------------------*)
    _FileWrite( bExecute:= FALSE );
    _FileWrite.sNetId    := '';  // local               
    _FileWrite.hFile     := _FileOpen.hFile;       
    _FileWrite.pWriteBuff:= ADR(_DataBuffer);
    _FileWrite.cbWriteLen:= _DataLength;
    _FileWrite.bExecute  := TRUE;
    _FileWrite.tTimeout  := Tc2_System.DEFAULT_ADS_TIMEOUT;
  END_IF

  (*-- ACTION ------------------------------------------------------------------------------------------------------------------*)
  _FileWrite();

  (*-- TRANSITION --------------------------------------------------------------------------------------------------------------*)
  IF (_FileWrite.bBusy = FALSE)
  THEN
    _FileSize  := _FileSize + _FileWrite.cbWrite;
    _WriteState:= E_TraceWriteStates.CloseSize;
  END_IF




(********************************************************************************************************************************)
(** close due to max file size exceeded *****************************************************************************************)
E_TraceWriteStates.CloseSize:
  (*-- ENTRY -------------------------------------------------------------------------------------------------------------------*)
  IF (_WriteStateLast <> _WriteState)
  THEN
    _WriteStateLast:= _WriteState;
    _WriteTime     := F_GetTimeMsTick();
    (*-----------------------------------------------------------------------------------*)
    _FileClose( bExecute:= FALSE );
    _FileClose.sNetId  := '';  // local
    _FileClose.hFile   := _FileOpen.hFile;
    _FileClose.bExecute:= TRUE;
    _FileClose.tTimeout:= Tc2_System.DEFAULT_ADS_TIMEOUT;
  END_IF

  (*-- ACTION ------------------------------------------------------------------------------------------------------------------*)
  _FileClose();

  (*-- TRANSITION --------------------------------------------------------------------------------------------------------------*)
  IF (_FileClose.bBusy = FALSE)
  THEN
    _FileIndex:= _FileIndex + 1;
    _Opened   := FALSE;
    (*-- calculate maximum file open time -----------------------------------------------*)
    _Statistics.MaxFileOpenTime:= MAX( _Statistics.MaxFileOpenTime, F_GetTimeMsDiff(_FileTimeOpened)  );
    (*-- error --------------------------------------------------------------------------*)
    IF    (_FileClose.bError = TRUE)
    THEN
      _WriteState:= E_TraceWriteStates.Error;
    (*-- closing successful -------------------------------------------------------------*)
    ELSE
      _WriteState:= E_TraceWriteStates.CreateOpen;
    END_IF
  END_IF




(********************************************************************************************************************************)
(** add eof due to new date *****************************************************************************************************)
E_TraceWriteStates.EofDate:
  (*-- ENTRY -------------------------------------------------------------------------------------------------------------------*)
  IF (_WriteStateLast <> _WriteState)
  THEN
    _WriteStateLast:= _WriteState;
    _WriteTime     := F_GetTimeMsTick();
    (*-- create eof ---------------------------------------------------------------------*)
{warning disable C0139}
    M_CreateEof();   _DataLength;
{warning restore C0139}
    (*-----------------------------------------------------------------------------------*)
    _FileWrite( bExecute:= FALSE );
    _FileWrite.sNetId    := '';  // local               
    _FileWrite.hFile     := _FileOpen.hFile;       
    _FileWrite.pWriteBuff:= ADR(_DataBuffer);
    _FileWrite.cbWriteLen:= _DataLength;
    _FileWrite.bExecute  := TRUE;
    _FileWrite.tTimeout  := Tc2_System.DEFAULT_ADS_TIMEOUT;
  END_IF

  (*-- ACTION ------------------------------------------------------------------------------------------------------------------*)
  _FileWrite();

  (*-- TRANSITION --------------------------------------------------------------------------------------------------------------*)
  IF (_FileWrite.bBusy = FALSE)
  THEN
    _FileSize  := _FileSize + _FileWrite.cbWrite;
    _WriteState:= E_TraceWriteStates.CloseDate;
  END_IF




(********************************************************************************************************************************)
(** close due to new date *******************************************************************************************************)
E_TraceWriteStates.CloseDate:
  (*-- ENTRY -------------------------------------------------------------------------------------------------------------------*)
  IF (_WriteStateLast <> _WriteState)
  THEN
    _WriteStateLast:= _WriteState;
    _WriteTime     := F_GetTimeMsTick();
    (*-----------------------------------------------------------------------------------*)
    _FileClose( bExecute:= FALSE );
    _FileClose.sNetId  := '';  // local
    _FileClose.hFile   := _FileOpen.hFile;
    _FileClose.bExecute:= TRUE;
    _FileClose.tTimeout:= Tc2_System.DEFAULT_ADS_TIMEOUT;
  END_IF

  (*-- ACTION ------------------------------------------------------------------------------------------------------------------*)
  _FileClose();

  (*-- TRANSITION --------------------------------------------------------------------------------------------------------------*)
  IF (_FileClose.bBusy = FALSE)
  THEN
    _Opened:= FALSE;
    (*-- calculate maximum file open time -----------------------------------------------*)
    _Statistics.MaxFileOpenTime:= MAX( _Statistics.MaxFileOpenTime, F_GetTimeMsDiff(_FileTimeOpened)  );
    (*-- error --------------------------------------------------------------------------*)
    IF    (_FileClose.bError = TRUE)
    THEN
      _WriteState:= E_TraceWriteStates.Error;
    (*-- closing successful -------------------------------------------------------------*)
    ELSE
      _WriteState:= E_TraceWriteStates.HddUsage;
    END_IF
  END_IF




(********************************************************************************************************************************)
(** read current hdd usage ******************************************************************************************************)
E_TraceWriteStates.HddUsage:
  (*-- ENTRY -------------------------------------------------------------------------------------------------------------------*)
  IF (_WriteStateLast <> _WriteState)
  THEN
    _WriteStateLast:= _WriteState;
    _WriteTime     := F_GetTimeMsTick();
    (*-----------------------------------------------------------------------------------*)
    _HddUsage.Start( Drive:= _MainFolder );  // use drive letter from main folder
  END_IF

  (*-- ACTION ------------------------------------------------------------------------------------------------------------------*)

  (*-- TRANSITION --------------------------------------------------------------------------------------------------------------*)
  IF (_HddUsage.Busy = FALSE)
  THEN
    _HddUsageCount:= _HddUsageCount + 1;
    _HddStateLast := E_TraceHddUsageStates.Initialization;  // force re-entry and write message
    (*-------------------------------------------*)
    _WriteState:= E_TraceWriteStates.StartWork;
  END_IF




(********************************************************************************************************************************)
(** unknown *********************************************************************************************************************)
ELSE
  _WriteState:= E_TraceWriteStates.Initialization;
END_CASE




(********************************************************************************************************************************)
(** done ************************************************************************************************************************)
END_METHOD

// maximum file size in kilobytes
{attribute 'monitoring' := 'call'}
PROPERTY PUBLIC MaxFileSizeKB : WORD
GET
MaxFileSizeKB:= _MaxFileSizeKB;
END_GET
SET
_MaxFileSizeKB:= MaxFileSizeKB;
END_SET
END_PROPERTY

// HI = file is currently open
{attribute 'monitoring' := 'call'}
PROPERTY PUBLIC Opened : BOOL
GET
Opened:= _Opened;
END_GET
END_PROPERTY

// puts a new trace line into the current file
METHOD PUBLIC Put

(********************************************************************************************************************************)
VAR_INPUT
  MsgType               : E_DebugMsgType                   := E_DebugMsgType.ERROR;
  Instance              : POINTER TO BYTE                  := 0;     // pointer to string
  Text                  : POINTER TO BYTE                  := 0;     // pointer to string
END_VAR

(********************************************************************************************************************************)
VAR
  Entry                 : POINTER TO FB_TraceEntry         := 0;
END_VAR

(********************************************************************************************************************************)
(** check inputs ****************************************************************************************************************)
IF (Text = 0)
THEN
  RETURN;
END_IF




(********************************************************************************************************************************)
(** enough hdd space? ***********************************************************************************************************)
IF (_HddTooFull = TRUE)
THEN
  _HddFullMissed:= _HddFullMissed + 1;
  RETURN;
END_IF




(********************************************************************************************************************************)
(** fb ready? *******************************************************************************************************************)
IF (System.fbSystemTime.TIMESTR.wYear = 0)
THEN
  _Diag_InvalidDate:= _Diag_InvalidDate + 1;
  RETURN;
END_IF




(********************************************************************************************************************************)
(** space in fifo available? ****************************************************************************************************)
IF (_FifoFillLevel >= FIFO_SIZE)
THEN
  _Diag_FifoFull:= _Diag_FifoFull + 1;
  RETURN;
END_IF




(********************************************************************************************************************************)
(** create entry ****************************************************************************************************************)
Entry:= __NEW( FB_TraceEntry( DateTime   := System.fbSystemTime.TIMESTR,
                              TaskCounter:= _TaskCounter + 1,
                             xMsgType    := MsgType,
                             xInstance   := Instance,  // leading x in the name:
                              Text       := Text  ) ); // Beckhoff SUPPORTCH-29439
IF   (Entry        = 0)      THEN  _Diag_NoMemory:= _Diag_NoMemory + 1;  RETURN;
ELSIF(Entry^.Valid = FALSE)  THEN  _Diag_NoEntry := _Diag_NoEntry  + 1;  __DELETE(Entry);  RETURN;
END_IF

_TaskCounter:= _TaskCounter + 1;





(********************************************************************************************************************************)
(** put into fifo ***************************************************************************************************************)
_Fifo[_FifoInput]:= Entry;

_FifoInput:= _FifoInput + 1;
IF(_FifoInput >= FIFO_SIZE)
THEN
  _FifoInput:= 0;
END_IF

_FifoFillLevel:= _FifoFillLevel + 1;




(********************************************************************************************************************************)
(** update statistics ***********************************************************************************************************)
_Statistics.PutCounter      := _Statistics.PutCounter  + 1;
_Statistics.MaxFifoFillLevel:= MAX(_Statistics.MaxFifoFillLevel, _FifoFillLevel);




(********************************************************************************************************************************)
(** done ************************************************************************************************************************)
END_METHOD

// diagnosis & statisticals
{attribute 'monitoring' := 'call'}
PROPERTY PUBLIC Statistics : I_TraceHandlerStatistics
GET
Statistics:= _Statistics;
END_GET
END_PROPERTY

END_FUNCTION_BLOCK

// ---- 20_Product/10_BCF/10_Base/11_Com/01_Stringhandling/F_StringCopy.TcPOU
// concats a string
FUNCTION PUBLIC F_StringCopy : POINTER TO BYTE

(**************************************************************************************
 * 	Application		:	BoxControl Framework
 *	Revision		  :	$Revision: 461868 $
 *	Revision date	:	$Date: 1979-01-09 14:35:13 +0200 (Di., 09 Jan 1979) $
 *	Last changed by	:	$Author: b7lipim $
 *	URL				:	$URL: http://almscdc.swisslog.com/repo/SWPD/Development/BoxControlFramework/20_Release/branches/R1.x/01_Software/BCF/BCF/JumpStart/20_Product/10_BCF/10_Base/11_Com/12_DebugMsg/00_GVLs/DebugTextBlocks.TcGVL $
 *
 * ------------------------------------------------------------------------------------
 *	Copyright Swisslog [IP AG], Switzerland. All rights reserved.
 * 
 * ------------------------------------------------------------------------------------
 *	
 * 	Revision History: 
 *
 * VERSION DATE         INITIALS     DESCRIPTION
 * 0.0     DD.MM.YYYY   (name)       (explain customized modifications)
 *
 **************************************************************************************)

(********************************************************************************************************************************)
VAR_INPUT
  DestStart             : POINTER TO BYTE                  := 0;     // = ADR(MyString)                    -> start position to concat
  DestEnd               : POINTER TO BYTE                  := 0;     // = ADR(MyString) + SIZEOF(MyString) -> buffer/string end
  (*----------------------------------------------------------------------------------------------------------------------------*)
  Source                : POINTER TO BYTE                  := 0;     // string to be copied
END_VAR

(********************************************************************************************************************************)
VAR
  DestWork             : POINTER TO BYTE                  := 0;
END_VAR


(********************************************************************************************************************************)
(** check inputs ****************************************************************************************************************)
IF   (DestStart = 0)         THEN  F_StringCopy:= 0;          RETURN;
ELSIF(DestEnd   = 0)         THEN  F_StringCopy:= DestStart;  RETURN;
ELSIF(DestStart >= DestEnd)  THEN  F_StringCopy:= DestStart;  RETURN;
ELSIF(Source    = 0)         THEN  F_StringCopy:= DestStart;  RETURN;
END_IF

DestWork:= DestStart;




(********************************************************************************************************************************)
(** copy characters *************************************************************************************************************)
WHILE (Source^ <> 16#00)
DO
  (*-- end of buffer reached --------------------------------------------------------------------------------*)
  IF (DestWork >= DestEnd)
  THEN
    DestWork := DestEnd - SIZEOF(DestWork^); // _DestWork^ hier benutzen
    EXIT;
  END_IF

  (*-- copy character ---------------------------------------------------------------------------------------*)
  DestWork^:= Source^;

  (*-- keep copying -----------------------------------------------------------------------------------------*)
  DestWork:= DestWork + SIZEOF(DestWork^);
  Source  := Source   + SIZEOF(Source^   );

END_WHILE

DestWork^:= 16#00;  // add termination




(********************************************************************************************************************************)
(** done ************************************************************************************************************************)
F_StringCopy:= DestWork;

END_FUNCTION

// ---- 20_Product/10_BCF/10_Base/11_Com/01_Stringhandling/F_StringFromDatestruct.TcPOU
// converts structure TIMESTR to string 'YYYY-MM-DD'
FUNCTION PUBLIC F_StringFromDatestruct : POINTER TO BYTE

(**************************************************************************************
 * 	Application		:	BoxControl Framework
 *	Revision		  :	$Revision: 461868 $
 *	Revision date	:	$Date: 1979-01-09 14:35:13 +0200 (Di., 09 Jan 1979) $
 *	Last changed by	:	$Author: b7lipim $
 *	URL				:	$URL: http://almscdc.swisslog.com/repo/SWPD/Development/BoxControlFramework/20_Release/branches/R1.x/01_Software/BCF/BCF/JumpStart/20_Product/10_BCF/10_Base/11_Com/12_DebugMsg/00_GVLs/DebugTextBlocks.TcGVL $
 *
 * ------------------------------------------------------------------------------------
 *	Copyright Swisslog [IP AG], Switzerland. All rights reserved.
 * 
 * ------------------------------------------------------------------------------------
 *	
 * 	Revision History: 
 *
 * VERSION DATE         INITIALS     DESCRIPTION
 * 0.0     DD.MM.YYYY   (name)       (explain customized modifications)
 *
 **************************************************************************************)

(********************************************************************************************************************************)
VAR_INPUT
  DestStart             : POINTER TO BYTE                  := 0;     // = ADR(MyString)                    -> start position to concat
  DestEnd               : POINTER TO BYTE                  := 0;     // = ADR(MyString) + SIZEOF(MyString) -> buffer/string end
  (*----------------------------------------------------------------------------------------------------------------------------*)
  DateStruct            : TIMESTRUCT;
END_VAR

(********************************************************************************************************************************)
VAR
  DestWork             : POINTER TO BYTE                  := 0;
END_VAR


(********************************************************************************************************************************)
(** check inputs ****************************************************************************************************************)
IF   (DestStart = 0)         THEN  F_StringFromDatestruct:= 0;          RETURN;
ELSIF(DestEnd   = 0)         THEN  F_StringFromDatestruct:= DestStart;  RETURN;
ELSIF(DestStart >= DestEnd)  THEN  F_StringFromDatestruct:= DestStart;  RETURN;
END_IF

DestWork:= DestStart;




(********************************************************************************************************************************)
(** convert *********************************************************************************************************************)
DestWork:= F_StringFromWord( DestStart:= DestWork,  DestEnd:= DestEnd,  Value:= DateStruct.wYear,   Length:= 4  );
DestWork:= F_StringCopy    ( DestStart:= DestWork,  DestEnd:= DestEnd,  Source:= ADR('-')  );
DestWork:= F_StringFromWord( DestStart:= DestWork,  DestEnd:= DestEnd,  Value:= DateStruct.wMonth,  Length:= 2  );
DestWork:= F_StringCopy    ( DestStart:= DestWork,  DestEnd:= DestEnd,  Source:= ADR('-')  );
DestWork:= F_StringFromWord( DestStart:= DestWork,  DestEnd:= DestEnd,  Value:= DateStruct.wDay,    Length:= 2  );




(********************************************************************************************************************************)
(** done ************************************************************************************************************************)
F_StringFromDatestruct:= DestWork;

END_FUNCTION

// ---- 20_Product/10_BCF/10_Base/11_Com/01_Stringhandling/F_StringFromWord.TcPOU
// converts word to string with specific length (adds zeros)
FUNCTION PUBLIC F_StringFromWord : POINTER TO BYTE

(**************************************************************************************
 * 	Application		:	BoxControl Framework
 *	Revision		  :	$Revision: 461868 $
 *	Revision date	:	$Date: 1979-01-09 14:35:13 +0200 (Di., 09 Jan 1979) $
 *	Last changed by	:	$Author: b7lipim $
 *	URL				:	$URL: http://almscdc.swisslog.com/repo/SWPD/Development/BoxControlFramework/20_Release/branches/R1.x/01_Software/BCF/BCF/JumpStart/20_Product/10_BCF/10_Base/11_Com/12_DebugMsg/00_GVLs/DebugTextBlocks.TcGVL $
 *
 * ------------------------------------------------------------------------------------
 *	Copyright Swisslog [IP AG], Switzerland. All rights reserved.
 * 
 * ------------------------------------------------------------------------------------
 *	
 * 	Revision History: 
 *
 * VERSION DATE         INITIALS     DESCRIPTION
 * 0.0     DD.MM.YYYY   (name)       (explain customized modifications)
 *
 **************************************************************************************)

(********************************************************************************************************************************)
VAR_INPUT
  DestStart             : POINTER TO BYTE                  := 0;     // = ADR(MyString)                    -> start position to concat
  DestEnd               : POINTER TO BYTE                  := 0;     // = ADR(MyString) + SIZEOF(MyString) -> buffer/string end
  (*----------------------------------------------------------------------------------------------------------------------------*)
  Value                 : WORD                             := 0;     // value to convert
  Length                : BYTE                             := 0;     // minimum string length (may be left stuffed with zeros)
END_VAR

(********************************************************************************************************************************)
VAR
  DestWork              : POINTER TO BYTE                  := 0;
  (*----------------------------------------------------------------------------------------------------------------------------*)
  Result                : STRING[7]                        := '';
  Size                  : WORD                             := 0;
  Stuff                 : WORD                             := 0;
END_VAR


(********************************************************************************************************************************)
(** check inputs ****************************************************************************************************************)
IF   (DestStart = 0)         THEN  F_StringFromWord:= 0;          RETURN;
ELSIF(DestEnd   = 0)         THEN  F_StringFromWord:= DestStart;  RETURN;
ELSIF(DestStart >= DestEnd)  THEN  F_StringFromWord:= DestStart;  RETURN;
END_IF

DestWork:= DestStart;




(********************************************************************************************************************************)
(** convert *********************************************************************************************************************)
Result:= WORD_TO_STRING(Value);
Size  := INT_TO_WORD( LEN(Result) );




(********************************************************************************************************************************)
(** stuff? **********************************************************************************************************************)
IF (Size < Length)
THEN
  Stuff:= Length - Size;
  (*-----------------------------------------------------------------*)
  WHILE(Stuff > 0)
  DO
    Stuff:= Stuff - 1;
    (*-------------------------------------------*)
    IF (DestWork >= DestEnd)
    THEN
      DestWork := DestEnd - SIZEOF(DestWork^); // _DestWork^ hier benutzen
      DestWork^:= 16#00;
      DestWork := DestEnd;
      EXIT;
    END_IF
    (*-- add '0' --------------------------------*)
    DestWork^:= 16#30;
    DestWork := DestWork + SIZEOF(DestWork^);
  END_WHILE
END_IF




(********************************************************************************************************************************)
(** copy characters *************************************************************************************************************)
DestWork:= F_StringCopy( DestStart:= DestWork,
                         DestEnd  := DestEnd,
                         Source   := ADR(Result)  );




(********************************************************************************************************************************)
(** done ************************************************************************************************************************)
F_StringFromWord:= DestWork;

END_FUNCTION

// ---- 20_Product/10_BCF/10_Base/11_Com/01_Stringhandling/F_StringFromTimestruct.TcPOU
// converts structure TIMESTR to string 'hh.mm.ss.mmm'
FUNCTION PUBLIC F_StringFromTimestruct : POINTER TO BYTE
(**************************************************************************************
 * 	Application		:	BoxControl Framework
 *	Revision		  :	$Revision: 461868 $
 *	Revision date	:	$Date: 1979-01-09 14:35:13 +0200 (Di., 09 Jan 1979) $
 *	Last changed by	:	$Author: b7lipim $
 *	URL				:	$URL: http://almscdc.swisslog.com/repo/SWPD/Development/BoxControlFramework/20_Release/branches/R1.x/01_Software/BCF/BCF/JumpStart/20_Product/10_BCF/10_Base/11_Com/12_DebugMsg/00_GVLs/DebugTextBlocks.TcGVL $
 *
 * ------------------------------------------------------------------------------------
 *	Copyright Swisslog [IP AG], Switzerland. All rights reserved.
 * 
 * ------------------------------------------------------------------------------------
 *	
 * 	Revision History: 
 *
 *  VERSION DATE         INITIALS     DESCRIPTION
 *  0.0     DD.MM.YYYY   (name)       (explain customized modifications)
 *
 **************************************************************************************)

(********************************************************************************************************************************)
VAR_INPUT
  DestStart             : POINTER TO BYTE                  := 0;     // = ADR(MyString)                    -> start position to concat
  DestEnd               : POINTER TO BYTE                  := 0;     // = ADR(MyString) + SIZEOF(MyString) -> buffer/string end
  (*----------------------------------------------------------------------------------------------------------------------------*)
  TimeStruct            : TIMESTRUCT;
  ShowMs                : BOOL                             := FALSE; // HI = shows milliseconds
END_VAR

(********************************************************************************************************************************)
VAR
  DestWork             : POINTER TO BYTE                  := 0;
END_VAR


(********************************************************************************************************************************)
(** check inputs ****************************************************************************************************************)
IF   (DestStart = 0)         THEN  F_StringFromTimestruct:= 0;          RETURN;
ELSIF(DestEnd   = 0)         THEN  F_StringFromTimestruct:= DestStart;  RETURN;
ELSIF(DestStart >= DestEnd)  THEN  F_StringFromTimestruct:= DestStart;  RETURN;
END_IF

DestWork:= DestStart;




(********************************************************************************************************************************)
(** convert *********************************************************************************************************************)
DestWork:= F_StringFromWord( DestStart:= DestWork,  DestEnd:= DestEnd,  Value:= TimeStruct.wHour,    Length:= 2  );
DestWork:= F_StringCopy    ( DestStart:= DestWork,  DestEnd:= DestEnd,  Source:= ADR(':')  );
DestWork:= F_StringFromWord( DestStart:= DestWork,  DestEnd:= DestEnd,  Value:= TimeStruct.wMinute,  Length:= 2  );
DestWork:= F_StringCopy    ( DestStart:= DestWork,  DestEnd:= DestEnd,  Source:= ADR(':')  );
DestWork:= F_StringFromWord( DestStart:= DestWork,  DestEnd:= DestEnd,  Value:= TimeStruct.wSecond,  Length:= 2  );

IF(ShowMs = TRUE)
THEN
  DestWork:= F_StringCopy    ( DestStart:= DestWork,  DestEnd:= DestEnd,  Source:= ADR(':')  );
  DestWork:= F_StringFromWord( DestStart:= DestWork,  DestEnd:= DestEnd,  Value:= TimeStruct.wMilliseconds,  Length:= 3  );
END_IF




(********************************************************************************************************************************)
(** done ************************************************************************************************************************)
F_StringFromTimestruct:= DestWork;

END_FUNCTION

// ---- 20_Product/10_BCF/10_Base/11_Com/02_Timings/F_GetTimeMsTick.TcPOU
// returns a timestamp (milliseconds)
FUNCTION PUBLIC F_GetTimeMsTick : TIME
(**************************************************************************************
 * 	Application		:	BoxControl Framework
 *	Revision		  :	$Revision: 461868 $
 *	Revision date	:	$Date: 1979-01-09 14:35:13 +0200 (Di., 09 Jan 1979) $
 *	Last changed by	:	$Author: b7lipim $
 *	URL				:	$URL: http://almscdc.swisslog.com/repo/SWPD/Development/BoxControlFramework/20_Release/branches/R1.x/01_Software/BCF/BCF/JumpStart/20_Product/10_BCF/10_Base/11_Com/12_DebugMsg/00_GVLs/DebugTextBlocks.TcGVL $
 *
 * ------------------------------------------------------------------------------------
 *	Copyright Swisslog [IP AG], Switzerland. All rights reserved.
 * 
 * ------------------------------------------------------------------------------------
 *	
 * 	Revision History: 
 *
 *  VERSION DATE         INITIALS     DESCRIPTION
 *  0.0     DD.MM.YYYY   (name)       (explain customized modifications)
 *
 **************************************************************************************)

(********************************************************************************************************************************)
VAR_INPUT
END_VAR

(********************************************************************************************************************************)
VAR
END_VAR


(********************************************************************************************************************************)
(** done ************************************************************************************************************************)
F_GetTimeMsTick:= TIME();

END_FUNCTION

// ---- 20_Product/10_BCF/10_Base/11_Com/02_Timings/F_GetTimeMsDiff.TcPOU
// returns a timedifference (in milliseconds) from TimeMsTick to now
FUNCTION PUBLIC F_GetTimeMsDiff : TIME
(**************************************************************************************
 * 	Application		:	BoxControl Framework
 *	Revision		  :	$Revision: 461868 $
 *	Revision date	:	$Date: 1979-01-09 14:35:13 +0200 (Di., 09 Jan 1979) $
 *	Last changed by	:	$Author: b7lipim $
 *	URL				:	$URL: http://almscdc.swisslog.com/repo/SWPD/Development/BoxControlFramework/20_Release/branches/R1.x/01_Software/BCF/BCF/JumpStart/20_Product/10_BCF/10_Base/11_Com/12_DebugMsg/00_GVLs/DebugTextBlocks.TcGVL $
 *
 * ------------------------------------------------------------------------------------
 *	Copyright Swisslog [IP AG], Switzerland. All rights reserved.
 * 
 * ------------------------------------------------------------------------------------
 *	
 * 	Revision History: 
 *
 *  VERSION DATE         INITIALS     DESCRIPTION
 *  0.0     DD.MM.YYYY   (name)       (explain customized modifications)
 *
 **************************************************************************************)

(********************************************************************************************************************************)
VAR_INPUT
  TimeMsTick            : TIME                             := T#0S;
END_VAR

(********************************************************************************************************************************)
VAR
END_VAR


(********************************************************************************************************************************)
(** done ************************************************************************************************************************)
F_GetTimeMsDiff:= F_GetTimeMsTick() - TimeMsTick;

END_FUNCTION

